// TIA Portal V20 export
TYPE "typeDataFromSafety"
// stored: Access Published, IsFailsafeCompliant true, Namespace Safety
   STRUCT
      devicesSummary { ExternalWritable := 'False'} : "Safety.typeDevicesStatusSummary";   // General safety status of devices
      mainOp { ExternalWritable := 'False'} : "Safety.typeMainOpMode";   // Main Op State
      pHmi { ExternalWritable := 'False'} : "Safety.typePhmi";
      scsMode { ExternalWritable := 'False'} : "Safety.typeScsMode";   // SCS Mode
      rcMode1 { ExternalWritable := 'False'} : "Safety.typeRollChangeMode";   // Top Roll Change State
      rcMode2 { ExternalWritable := 'False'} : "Safety.typeRollChangeMode";   // Btm Roll Change State
      eStopStatus { ExternalWritable := 'False'} : "Safety.typeEstopStatus";   // E Stop Pressed
      fDoorSwitchStatus { ExternalWritable := 'False'} : "Safety.typeFDoorSwitchStatus";   // F Door Open Status
      fDoorCoilStatus { ExternalWritable := 'False'} : "Safety.typeFDoorUnlockOutput";   // F Door Unlock Cmd Status
      Zone1SafetyMainOpEnable { ExternalWritable := 'False'} : "Safety.typeSafetyOperationEnable";   // Zone1 Main Operation Enable
      Zone1SafetySubOpEnable { S7_SetPoint := 'True'} : "Safety.typeSafetyOperationEnable";   // Zone1 Sub Operation Enable
      Zone2SafetyOpEnable { ExternalWritable := 'False'} : "Safety.typeSafetyOperationEnable";   // Zone2 Operation Enable
      Zone3SafetyOpEnable { ExternalWritable := 'False'} : "Safety.typeSafetyOperationEnable";   // Zone3 Operation Enable
      eStopZone1 { ExternalWritable := 'False'} : "Safety.typeEstopFunction";   // Safety status of estop button in Zone.1
      eStopZone2 { ExternalWritable := 'False'} : "Safety.typeEstopFunction";   // Safety status of estop button in Zone.2
      eStopZone3 { ExternalWritable := 'False'} : "Safety.typeEstopFunction";   // Safety status of estop button in Zone.3
      statusZone1 { ExternalWritable := 'False'} : "Safety.typeSafetyZoneStatus";   // Status of safety zone
      statusZone2 { ExternalWritable := 'False'} : "Safety.typeSafetyZoneStatus";   // Status of safety zone
      statusZone3 { ExternalWritable := 'False'} : "Safety.typeSafetyZoneStatus";   // Status of safety zone
      fDoorDrive : "Safety.typeFDoorFunction";
      driveStatus : "Safety.typeSafetyDriveStatus";
      SafetySensor { ExternalWritable := 'False'} : "Safety.typeSafetySensor";
      FeedbackFault { ExternalWritable := 'False'} : "Safety.typeFeedbackFault";
      AllEstopsOK { ExternalWritable := 'False'} : Bool;   // E Stop On Station All Ok
      allEstopButtonsOK : Bool;
      AllEstopsOKfromOther : Bool;   // E Stop On Other Station All Ok
      AllFdoorClose { ExternalWritable := 'False'} : Bool;   // F Door All Closed
      AllSFDoorOpen { ExternalWritable := 'False'} : Bool;   // F Door Single Open
      AnyNoMFDoorOpen { ExternalWritable := 'False'} : Bool;   // F Door No Multi Open
      safetyReleasedAllSafetyZones { ExternalWritable := 'False'} : Bool := false;   // All safety zones are released
      ackRequiredAnySafetyZone { ExternalWritable := 'False'} : Bool := false;   // At least one safety zone requires an acknowledge
      ackOP_changeRequired { ExternalWritable := 'False'} : Bool := false;   // ACK_OP is waiting for value change
      ackOperatorControlCondition : Bool;   // Ack Hmi Oprating Possible
      doorBoxAllReset : Bool;   // Combine All Door Box Reset Button
      totalSafetyReset { ExternalAccessible := 'False'; ExternalVisible := 'False'; ExternalWritable := 'False'} : Bool;   // Combine All Reset Trigger
      zone1DoorOpenRequest : Bool;   // Zone 1 Door Open Request
      zone2DoorOpenRequest : Bool;   // Zone 2 Door Open Request
      zone3DoorOpenRequest : Bool;   // Zone 3 Door Open Request
      zone1DriveAckReq : Bool;   // Zone 1 Safety Fault Ack Request
      zone2DriveAckReq : Bool;   // Zone 2 Safety Fault Ack Request
      zone3DriveAckReq : Bool;   // Zone 3 Safety Fault Ack Request
      noSafetyFault : Bool;   // All Zone No Safety Fault
      ConnectionBoxID { ExternalWritable := 'False'} : Int := 0;   // PHmi Connection Box ID
      BA60jrPPLeftDoorForcedOpen : Bool;   // BA060 JR P&P Left Door Forced Open
      BA060STOP : Bool;   // In Execute Stop Request From BA060
      BA60LightCurtainMuttingRequest : Bool;   // Light Curtain Mutting Request To BA060
      BA60LightCurtainDetect : Bool;   // BA060 Light Curtain Detect
      BA60RequestForEntry : Bool;   // Sepa Gripper Entry For Request From BA060
      BA60ExternalDoorOpen : Bool;
      BA60jrPPLeftDoorNormalOpen : Bool;   // BA060 JR P&P Left Door Normal Open
      PhmiConnectedToBA60 : Bool;
      PhmiEnableToBA60 : Bool;
      HmiEnableToBA60 : Bool;
      BA40CathodeCoverClose : Bool;
      BA40AnodeCoverClose : Bool;
      BA60Stacker2LightCurtainDetect : Bool;
      BA60Stacker2MaintanceDoorOpen : Bool;
      SS1TimeExtension : Bool;
      EnableServoAck : Bool;
      SetupModeFault : Bool;
      CathodeCoverSensorFault : Bool;
      AnodeCoverSensorFault : Bool;
      Door02UnlockPB : Bool;
      Door03UnlockPB : Bool;
      Door04UnlockPB : Bool;
      Door05UnlockPB : Bool;
      BA10 { ExternalWritable := 'False'} : "Safety.typeDataFlinkUsed";
      BA15 { ExternalWritable := 'False'} : "Safety.typeDataFlinkUsed";
      BA40 { ExternalWritable := 'False'} : "Safety.typeDataFlinkUsed";
      BA60 { ExternalWritable := 'False'} : "Safety.typeDataFlinkUsed";
      cvCoverStatus { ExternalWritable := 'False'} : "Safety.typeCvCoverStatus";
      hotWireCutterStatus { ExternalWritable := 'False'} : "Safety.typeHotWireCutter";
      fDoorUnwinderTopDoorOpenWarning { ExternalWritable := 'False'} : Bool;
      fDoorUnwinderBtmDoorOpenWarning { ExternalWritable := 'False'} : Bool;
      PhmiForcedDisconnection : Bool;
      CathodeConveyorCoverClosedCheck : Bool;
      AnodeConveyorCoverClosedCheck : Bool;
      FDoorForcedOpenStatus : "Safety.typeSafetyForcedDoorOpen";
   END_STRUCT;
END_TYPE
